// Mitsubishi GX Works2 project: LAB 1   PLC: FX1N/FX1NC

PROGRAM MAIN
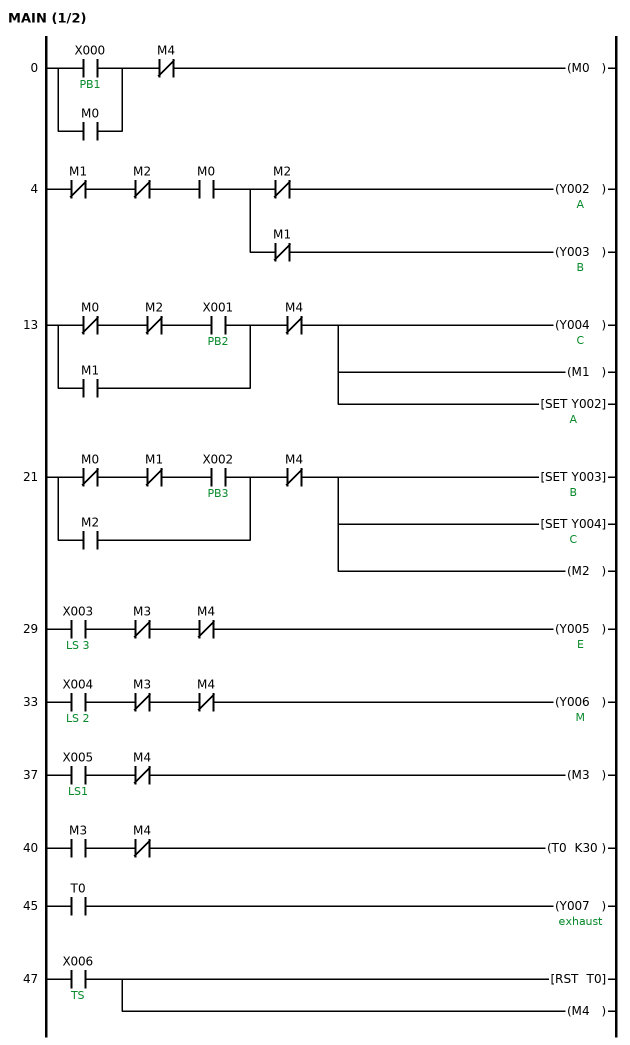
0     LD      X000  ; PB1
      OR      M0
      ANI     M4
      OUT     M0
4     LDI     M1
      ANI     M2
      AND     M0
      MPS
      ANI     M2
      OUT     Y002  ; A
      MPP
      ANI     M1
      OUT     Y003  ; B
13    LDI     M0
      ANI     M2
      AND     X001  ; PB2
      OR      M1
      ANI     M4
      OUT     Y004  ; C
      OUT     M1
      SET     Y002  ; A
21    LDI     M0
      ANI     M1
      AND     X002  ; PB3
      OR      M2
      ANI     M4
      SET     Y003  ; B
      SET     Y004  ; C
      OUT     M2
29    LD      X003  ; LS 3
      ANI     M3
      ANI     M4
      OUT     Y005  ; E
33    LD      X004  ; LS 2
      ANI     M3
      ANI     M4
      OUT     Y006  ; M
37    LD      X005  ; LS1
      ANI     M4
      OUT     M3
40    LD      M3
      ANI     M4
      OUT     T0 K30
45    LD      T0
      OUT     Y007  ; exhaust
47    LD      X006  ; TS
      RST     T0
      OUT     M4
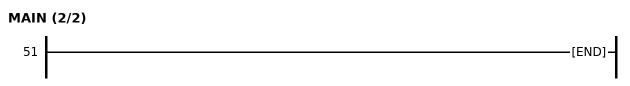
51    END
END_PROGRAM
